ABB RobotStudio station: Solution maximum speed.rspag

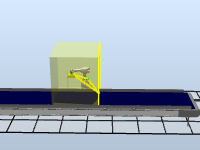
--- station ---
Station Solution1 (saved by RobotStudio 6.8.8148.134)
Controller System1, task T_ROB1: task frame (RAPID world) sits at (5535.63, 748.67, 709.58) mm in the station
Controller System1
  mechanical unit ROB_1: IRB1600_10_145__01, 6 joints, base frame (480.91, -394.38, -359.58) mm, rotated rx 0 ry 0 rz 90 deg
  mechanical unit CNV1: ?, 1 joints, base frame (0, 0, 0) mm
Layout (positions relative to the parent item):
  - bin mover_3 [smart component, from libraries\bin mover.rslib] at (-500, 0, 0) mm
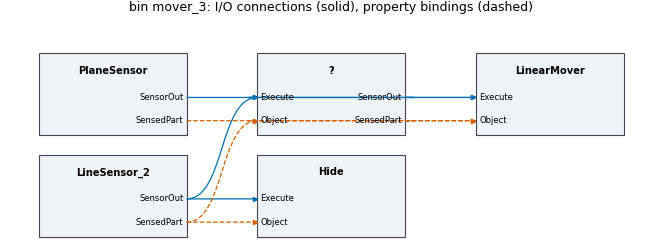
      connections:
        ?.SensorOut -> LinearMover.Execute
        PlaneSensor.SensorOut -> LinearMover.Execute
        ?.SensorOut -> ?.Execute
        LineSensor_2.SensorOut -> ?.Execute
        LineSensor_2.SensorOut -> Hide.Execute
        ?.SensedPart => LinearMover.Object
        PlaneSensor.SensedPart => LinearMover.Object
        ?.SensedPart => ?.Object
        LineSensor_2.SensedPart => ?.Object
        LineSensor_2.SensedPart => Hide.Object
    - LinearMover [smart component, from Components\LinearMover.rslib] at (6663.26, 677.27, 1050.93) mm, rotated rx 180 ry 0 rz 90 deg
        properties: Object=(none); Direction=[0 0 -1]; Speed=8; Reference=Global; ReferenceObject=(none)
    - PlaneSensor [smart component, from Components\PlaneSensor.rslib]
        properties: Origin=[7.419145 0.146999 1.42]; Axis1=[0 0 -1.35]; Axis2=[0 0.4 0]; SensedPart=(none)
      - _sensorPart_ [part, from libraries\bin mover.rslib]
    - LineSensor_2 [smart component, from Components\LineSensor.rslib]
        properties: Start=[7.369145 0.346999 0.008]; End=[7.369145 0.346999 0.123]; Radius=0.09; SensedPart=(none); SensedPoint=[0 0 0]
      - _sensorPart_ [part, from libraries\bin mover.rslib]
    - Hide [smart component, from Components\Hide.rslib]
        properties: Object=(none)
  - bin1_2 [part, from libraries\bin1.rslib] at (6733.74, 347, -12) mm
  - conveyor 1 [part] at (0, -1500, -4460) mm, rotated rx 90 ry 0 rz 90 deg
  - Suction gripper 18cm [smart component] at (6727.84, 418.35, 1386.5) mm, rotated rx 180 ry 0 rz -90 deg
      signals: DI do1
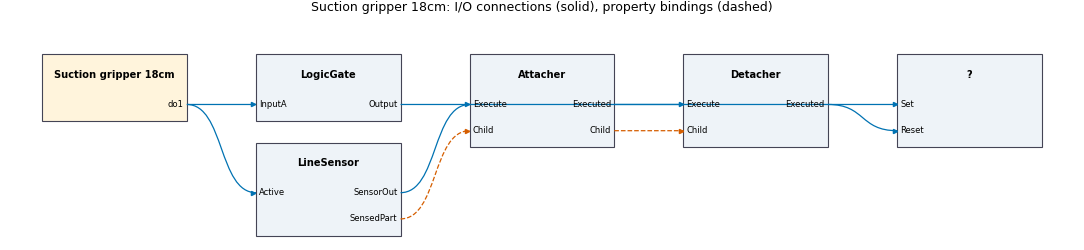
      connections:
        Suction gripper 18cm.do1 -> LogicGate.InputA
        Suction gripper 18cm.do1 -> LineSensor.Active
        LogicGate.Output -> Detacher.Execute
        LineSensor.SensorOut -> Attacher.Execute
        Attacher.Executed -> ?.Set
        Detacher.Executed -> ?.Reset
        LineSensor.SensedPart => Attacher.Child
        Attacher.Child => Detacher.Child
    - Attacher [smart component, from Components\Attacher.rslib]
        properties: Parent=Suction_gripper 18cm; Flange=0; Child=Yellow block; Mount=false; Offset=[0 0 0]; Orientation=[0 0 0]
    - LogicGate [smart component, from Components\LogicGate.rslib]
        properties: Operator=NOT; Delay=0
    - LineSensor [smart component, from Components\LineSensor.rslib] at (7150.29, 306.47, 1168.39) mm, rotated rx 180 ry 0 rz 90 deg
        properties: Start=[-0.30577796087058 -7.14894421240012 1.16938863540814]; End=[-0.305777964813962 -7.14894420825673 1.13938863540814]; Radius=0.09; SensedPart=Yellow block; SensedPoint=[6.26593994140625 0.816847717285156 1.04397839355469]
      - _sensorPart_ [part]
    - Detacher [smart component, from Components\Detacher.rslib]
        properties: Child=Yellow block; KeepPosition=true
  - Suction_gripper 18cm [mechanism, from libraries\Suction_gripper_18cm.rslib] at (6727.84, 418.35, 1471.5) mm, rotated rx 180 ry 0 rz -90 deg
  - IRB1600_10_145__01 [mechanism, from Robots\IRB1600_10_145_G_01.rslib] at (6016.55, 235.44, 350) mm, rotated rx 0 ry 0 rz 90 deg; joint values [-1.3191, -0.0222, 0.0219, 0, 1.5711, -1.3191] (rad or m)
  - 输送链 [conveyor]
    - Conveyor cover [part] at (-300, 0, 14) mm
    - Yellow block [part] at (0, -475.41, 0) mm
    - 传送带对象_17 [conveyorobject] at (9408.59, 748.67, 709.58) mm
      - Yellow block [part] at (-796.77, -1777.48, -1495.2) mm
    - 传送带对象_18 [conveyorobject] at (6708.59, 748.67, 709.58) mm
      - Yellow block [part] at (-792.91, -1777.35, -1495.7) mm
    - 传送带对象_19 [conveyorobject] at (4008.59, 748.67, 709.58) mm
      - Yellow block [part] at (-295.22, -1778.45, -145.75) mm
Attachment: Suction gripper 18cm is attached to Suction_gripper 18cm / Suction gripper 18cm
Attachment: Suction_gripper 18cm is attached to IRB1600_10_145__01 / Link6
Conveyor tracking 连接_2: unit CNV1, TravelOffset=3.7, QueueTrackDistance=0, StartWindowWidth=1.8, SyncSeparation=0, CountsPerMeter=10000
Station logic (signal -> signal, property => property):
  System1.do_attach -> Suction gripper 18cm.do1

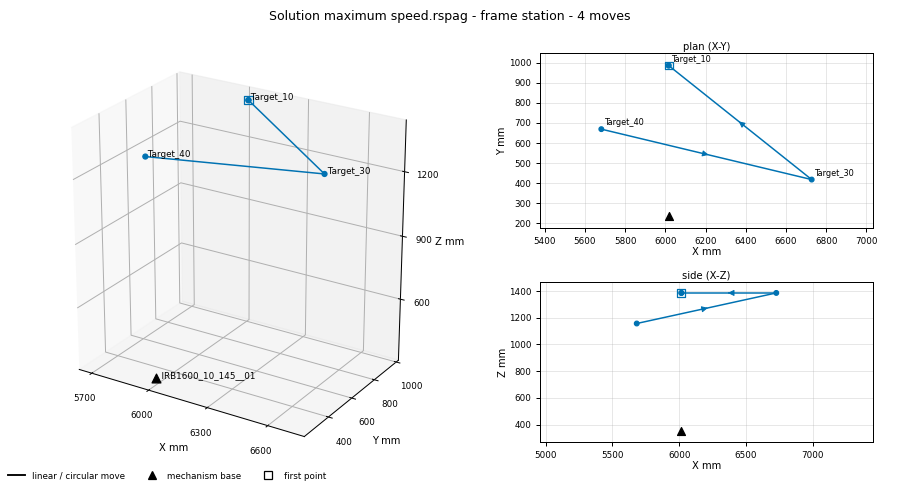
[picture p0: tool path of Solution maximum speed.rspag in frame station, 4 of 5 moves have a stored position in this frame; points joined in program order, loops and branches not executed]
--- Backups/System1/RAPID/TASK1/PROGMOD/CalibData.mod ---
MODULE CalibData
	TASK PERS wobjdata wobj_cnv1:=[FALSE,FALSE,"CNV1",[[0,0,0],[1,0,0,0]],[[0,0,0],[1,0,0,0]]];
	PERS tooldata Suction_gripper_18cm:=[TRUE,[[0,0,85],[1,0,0,0]],[1,[0,0,1],[1,0,0,0],0,0,0]];
ENDMODULE

--- Backups/System1/RAPID/TASK1/PROGMOD/Module1.mod ---
MODULE Module1
    VAR num y:=0;
	CONST robtarget Target_10:=[[480.915,236.77,676.92],[0,-0.707106781,0.707106781,0],[0,0,0,0],[9E+09,9E+09,9E+09,9E+09,9E+09,0]];
	CONST robtarget Target_20:=[[29.699626144,355.874016057,111.58001204],[0.000000002,0.707106781,-0.707106781,0.000000007],[0,-1,0,0],[9E+09,9E+09,9E+09,9E+09,9E+09,0]];
	CONST robtarget Target_30:=[[1192.207950487,-330.312717415,676.919992598],[0.000000021,0.707106781,-0.707106781,0.000000022],[-1,-1,-1,0],[9E+09,9E+09,9E+09,9E+09,9E+09,0]];
	CONST robtarget Target_40:=[[146.179414768,-79.610437519,447.822390714],[0.000000004,0.707106782,-0.70710678,0.000000059],[0,-1,0,0],[9E+09,9E+09,9E+09,9E+09,9E+09,0]];

    PROC main()
        ActUnit CNV1;

        WHILE 2>1 DO

            WaitWObj wobj_cnv1;
            Path_10;
            DropWObj wobj_cnv1;

        ENDWHILE
    ENDPROC
    PROC Path_10()
		MoveL Target_10,vmax,z0,Suction_gripper_18cm\WObj:=wobj0;
		MoveL Target_20,vmax,z10,Suction_gripper_18cm\WObj:=wobj_cnv1;
		Set do_attach;
		MoveL Target_40,vmax,z10,Suction_gripper_18cm\WObj:=wobj0;
		MoveL Target_30,vmax,fine,Suction_gripper_18cm\WObj:=wobj0;
		Reset do_attach;
		MoveL Target_10,vmax,z0,Suction_gripper_18cm\WObj:=wobj0;

    ENDPROC
ENDMODULE

--- Backups/System1/SYSPAR/EIO.cfg ---
EIO:CFG_1.0:6:1::
#
INDUSTRIAL_NETWORK:

      -Name "RobICI" -Label "RobICI Network"

      -Name "DeviceNet" -Label "DeviceNet Master/Slave Network" -Address "2"
#
ROBICI_DEVICE:

      -Name "CTM1" -TrustLevel "InternalDeviceTrustLevel"\
      -VendorName "ABB Robotics" -ProductName "DSQC2000"\
      -Label "Conveyor Tracking Device 1" -Address "0.0.0.0"
#
DEVICENET_INTERNAL_DEVICE:

      -Name "DN_Internal_Device" -VendorName "ABB Robotics"\
      -ProductName "DeviceNet Internal Slave Device"
#
EIO_SIGNAL:

      -Name "c1Counts" -SignalType "GI" -Device "CTM1"\
      -DeviceMap "Enc1:position"

      -Name "c1CountsPerSec" -SignalType "AI" -Device "CTM1"\
      -DeviceMap "Enc1:velocity"

      -Name "c1TrigVis" -SignalType "DO" -Device "CTM1" -Label "Trig X21 pin 5"\
      -DeviceMap "Digout1:Setpoint"

      -Name "c1TrigAutoMode" -SignalType "DO" -Device "CTM1"\
      -DeviceMap "Cam1:Connect"

      -Name "c1TrigAutoDist" -SignalType "GO" -Device "CTM1"\
      -DeviceMap "Cam1:Interval"

      -Name "c1TrigAutoEncNo" -SignalType "GO" -Device "CTM1"\
      -DeviceMap "Cam1Enc:DeviceNo"

      -Name "c1CntFromEnc" -SignalType "GI" -Device "CTM1"\
      -DeviceMap "Sync1Enc1:Value"

      -Name "c1SoftSync" -SignalType "DO" -Device "CTM1"\
      -DeviceMap "Sync1Enc1:SyncTrig"

      -Name "c1SpeedBandWidth" -SignalType "GI" -Device "CTM1"\
      -DeviceMap "e1_SpeedBandWidth:SetPoint"

      -Name "c1Position" -SignalType "AO" -MaxLog 21474.8 -MaxPhys 1\
      -MaxPhysLimit 1 -MaxBitVal 2147483647 -MinLog -21474.8 -MinPhys -1\
      -MinPhysLimit -1 -MinBitVal -2147483647 -Size 32

      -Name "c1Speed" -SignalType "AO" -MaxLog 21474.8 -MaxPhys 1\
      -MaxPhysLimit 1 -MaxBitVal 2147483647 -MinLog -21474.8 -MinPhys -1\
      -MinPhysLimit -1 -MinBitVal -2147483647 -Size 32

      -Name "c1Connected" -SignalType "DO"

      -Name "c1NullSpeed" -SignalType "DO"

      -Name "c1PassStw" -SignalType "DO"

      -Name "c1NewObjStrobe" -SignalType "DO"

      -Name "c1WaitWObj" -SignalType "DO"

      -Name "c1DropWObj" -SignalType "DO" -Access "ALL"

      -Name "c1Rem1PObj" -SignalType "DO" -Access "All"

      -Name "c1RemAllPObj" -SignalType "DO" -Access "All"

      -Name "c1CntToEncStr" -SignalType "DO"

      -Name "c1PosInJobQ" -SignalType "DO" -Default 1

      -Name "c1ObjectsInQ" -SignalType "GO" -Size 8

      -Name "c1CntToEnc" -SignalType "GO" -Size 32

      -Name "do_attach" -SignalType "DO"

--- Backups/System1/SYSPAR/PROC.cfg ---
PROC:CFG_1.0:6:0::
#
CONVEYOR:

      -name "CNV1" -sensor_type "ICI" -use_sensor "ICI1" -adjustment_speed 850\
      -min_dist -1 -max_dist 20000 -correction_vector_ramp_length 5
#
CONVEYOR_ICI_SENSOR:

      -name "ICI1" -connected_signal "c1Connected" -position_signal "c1Position"\
      -velocity_signal "c1Speed" -position_count_signal "c1Counts"\
      -velocity_count_signal "c1CountsPerSec" -null_speed_signal "c1NullSpeed"\
      -wait_wobj_signal "c1WaitWObj" -drop_wobj_signal "c1DropWObj"\
      -rem_all_pobj_signal "c1RemAllPObj" -rem_one_pobj_signal "c1Rem1PObj"\
      -supervise_max_dist_off  -newobj_strobe "c1NewObjStrobe"\
      -count_to_enc_strobe "c1CntToEncStr" -obj_in_queue_signal "c1ObjectsInQ"\
      -count_from_enc "c1CntFromEnc" -count_to_enc "c1CntToEnc"\
      -StartWinWidth 1.8 -speed_filter_bandwidth "c1SpeedBandWidth"
